// TIA Portal V20 export
DATA_BLOCK "DB_UDI"   // DB44
// stored: MemoryReserve 100, Namespace PackedLine
   VAR
      PackedLine : Struct
         Upstream : Struct
            Conveyor : Array[_.minPackedLine.._.maxPackedLine] of Bool;
         END_STRUCT;
         DownstreamAcu : Struct
            Stop : Struct
               Conveyor : Array[_.minPackedLine.._.maxPackedLine] of Bool;
            END_STRUCT;
         END_STRUCT;
         Interlock : Struct
            Stop : Struct
               Conveyor : Array[_.minPackedLine.._.maxPackedLine] of Bool;
            END_STRUCT;
         END_STRUCT;
         Fault : Struct
            Stop : Struct
               Conveyor : Array[_.minPackedLine.._.maxPackedLine] of Bool;
            END_STRUCT;
         END_STRUCT;
         Transfer : Struct
            "B1.6.1" : Struct
               "Upstream Straight" : Bool;
               "Upstream Arm" : Bool;
            END_STRUCT;
         END_STRUCT;
      END_STRUCT;
   END_VAR
BEGIN
END_DATA_BLOCK
